// Mitsubishi GX Works2 project: Master_prog_VH_2604   PLC: Q00

// global labels: Global1
VAR_GLOBAL
  pumpFlag AT M40 : BOOL;
  alarmLightFlag : BOOL;
  magValve1Flag AT M42 : BOOL;
  magValve2Flag AT M43 : BOOL;
  magValve3Flag AT M44 : BOOL;
  Kp AT D2 : INT;
  Ti AT D3 : INT;
  Td AT D4 : INT;
  Tf AT D5 : INT;
  kFF AT D6 : INT;
  tFF AT D7 : INT;
  nFF AT D8 : INT;
  setpunkt_begrensning AT D9 : INT;  (* Bestemmer hvor mye setpunktet max kan øke hvert scan *)
  setpunkt AT D10 : INT;
  manU AT D11 : INT;
  nomU AT D12 : INT;
  manU_HMI AT D13 : INT;
  nomU_HMI AT D14 : INT;
  sepunkt AT D1001 : INT;  (* Ønsketsetpunkt *)
  setpunkt_rampe AT D1002 : INT;  (* Bruk denne for alarmsystemet, dette er det faktiske setpunktet! som er rampet opp *)
  to_slave AT D60 : INT;
  man AT M102 : BOOL;  (* Bestemmer man/auto modus *)
  rampPaa AT D15 : INT;  (* bestemmer om setpunkt rampes *)
END_VAR

// task Task_01 (event TRUE, interval 0, priority 31): com_interface
// task main_prog (event TRUE, interval 0, priority 31): main_prog
// user libraries (not included): PIDFERDIG

PROGRAM com_interface
(* structured ladder/FBD written out as ST: instructions are called as NAME(EN, inputs, outputs); _pN, _eN, _tN stand for wires *)
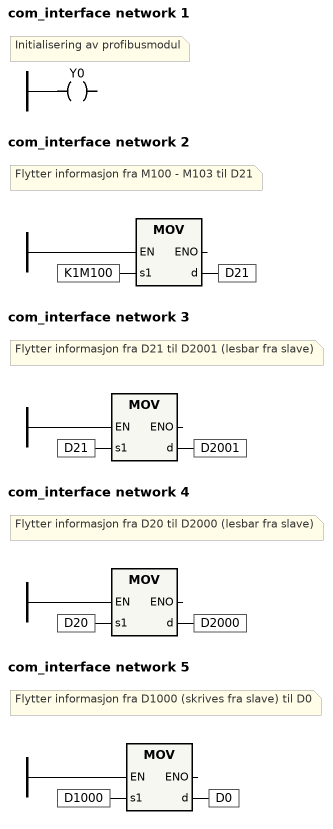
(* network 1 *)
(* Initialisering av profibusmodul *)
Y0 := TRUE;
(* network 2 *)
(* Flytter informasjon fra M100 - M103 til D21 *)
MOV(TRUE, K1M100, D21);
(* network 3 *)
(* Flytter informasjon fra D21 til D2001 (lesbar fra slave) *)
MOV(TRUE, D21, D2001);
(* network 4 *)
(* Flytter informasjon fra D20 til D2000 (lesbar fra slave) *)
MOV(TRUE, D20, D2000);
(* network 5 *)
(* Flytter informasjon fra D1000 (skrives fra slave) til D0 *)
MOV(TRUE, D1000, D0);
END_PROGRAM

PROGRAM main_prog
VAR
  to_slave : INT;
  from_slave : INT;
END_VAR
(* structured ladder/FBD written out as ST: instructions are called as NAME(EN, inputs, outputs); _pN, _eN, _tN stand for wires *)
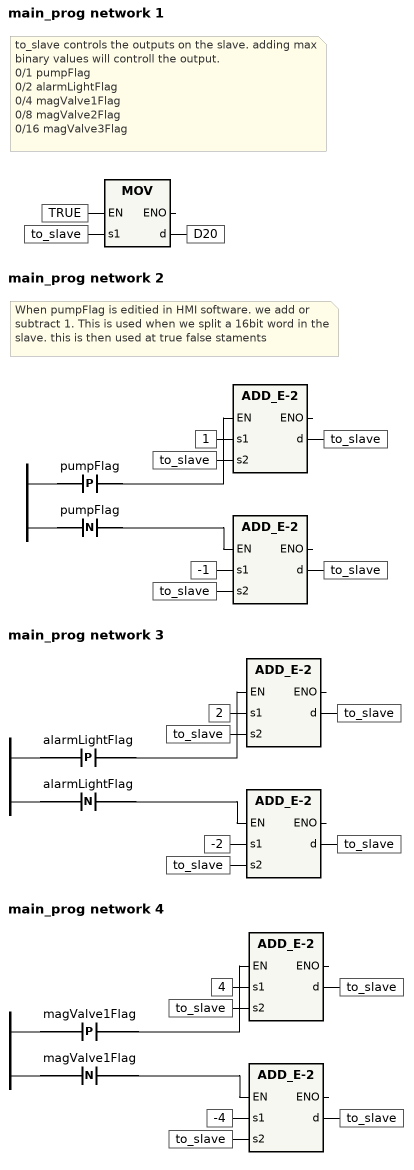
(* network 1 *)
(* to_slave controls the outputs on the slave. adding max binary values will controll the output.  /  / 0/1 pumpFlag / 0/2 alarmLightFlag / 0/4 magValve1Flag  / 0/8 magValve2Flag  / 0/16 magValve3Flag *)
MOV(TRUE, to_slave, D20);
(* network 2 *)
(* When pumpFlag is editied in HMI software. we add or subtract 1. This is used when we split a 16bit word in the slave. this is then used at true false staments *)
ADD_E(LDP(TRUE, pumpFlag), 1, to_slave, to_slave);
ADD_E(LDF(TRUE, pumpFlag), -1, to_slave, to_slave);
(* network 3 *)
ADD_E(LDP(TRUE, alarmLightFlag), 2, to_slave, to_slave);
ADD_E(LDF(TRUE, alarmLightFlag), -2, to_slave, to_slave);
(* network 4 *)
ADD_E(LDP(TRUE, magValve1Flag), 4, to_slave, to_slave);
ADD_E(LDF(TRUE, magValve1Flag), -4, to_slave, to_slave);
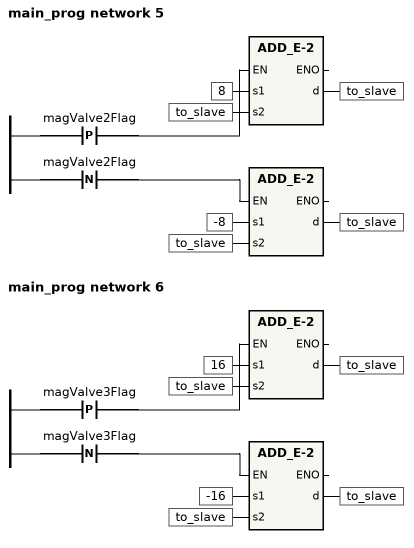
(* network 5 *)
ADD_E(LDP(TRUE, magValve2Flag), 8, to_slave, to_slave);
ADD_E(LDF(TRUE, magValve2Flag), -8, to_slave, to_slave);
(* network 6 *)
ADD_E(LDP(TRUE, magValve3Flag), 16, to_slave, to_slave);
ADD_E(LDF(TRUE, magValve3Flag), -16, to_slave, to_slave);
END_PROGRAM

PROGRAM Prossesverdier_kom
(* structured ladder/FBD written out as ST: instructions are called as NAME(EN, inputs, outputs); _pN, _eN, _tN stand for wires *)
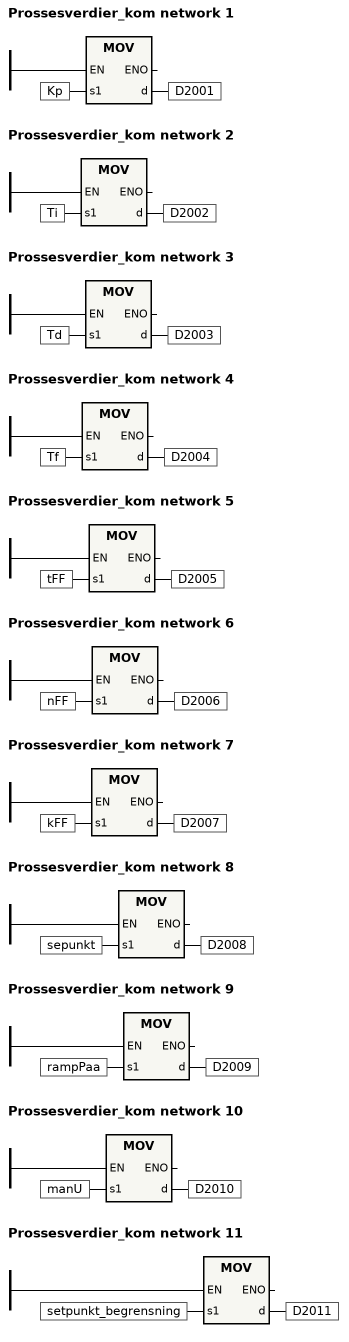
(* network 1 *)
MOV(TRUE, Kp, D2001);
(* network 2 *)
MOV(TRUE, Ti, D2002);
(* network 3 *)
MOV(TRUE, Td, D2003);
(* network 4 *)
MOV(TRUE, Tf, D2004);
(* network 5 *)
MOV(TRUE, tFF, D2005);
(* network 6 *)
MOV(TRUE, nFF, D2006);
(* network 7 *)
MOV(TRUE, kFF, D2007);
(* network 8 *)
MOV(TRUE, sepunkt, D2008);
(* network 9 *)
MOV(TRUE, rampPaa, D2009);
(* network 10 *)
MOV(TRUE, manU, D2010);
(* network 11 *)
MOV(TRUE, setpunkt_begrensning, D2011);
END_PROGRAM
